{attribute 'GeneratedUsingTerminal: EL5021-0000-0016'}
{attribute addProperty BoxType "EL5021-0000-0016"}
{attribute addProperty Id "EtcSlaveTerminalBaseENC_StatusAT %I*ENC_Status_1E2673DC16ENC_ControlAT %Q*ENC_Control_64DD586E6WcStateAT %I*WcState_9091E0EB2InfoDataAT %I*InfoData_32EB74EA10"}
{attribute addProperty CRC "1219258104"}
{attribute addProperty Size "34"}
TYPE EL5021_48AC66F8 EXTENDS EtcSlaveTerminalBase :
STRUCT
	{attribute addProperty Name "ENC_Status"}
	ENC_Status : ENC_Status_1E2673DC;
	{attribute addProperty Name "ENC_Control"}
	ENC_Control : ENC_Control_64DD586E;
	{attribute addProperty Name "WcState"}
	WcState : WcState_9091E0EB;
	{attribute addProperty Name "InfoData"}
	InfoData : InfoData_32EB74EA;
END_STRUCT
END_TYPE

(* stored: Version 1.2.0.0, ProductVersion 3.1.4024.9
   DUT EL5021_48AC66F8: Id {56ea7788-3792-4fdb-b25b-0c984b980b06} *)
